INTERFACE ITF_BaseHMILoggerElement_Command

END_INTERFACE

(* stored: Version 1.1.0.1
   Itf ITF_BaseHMILoggerElement_Command: Id {8a9d56ad-23ca-0251-2e0b-7f69bd8f3607} *)
